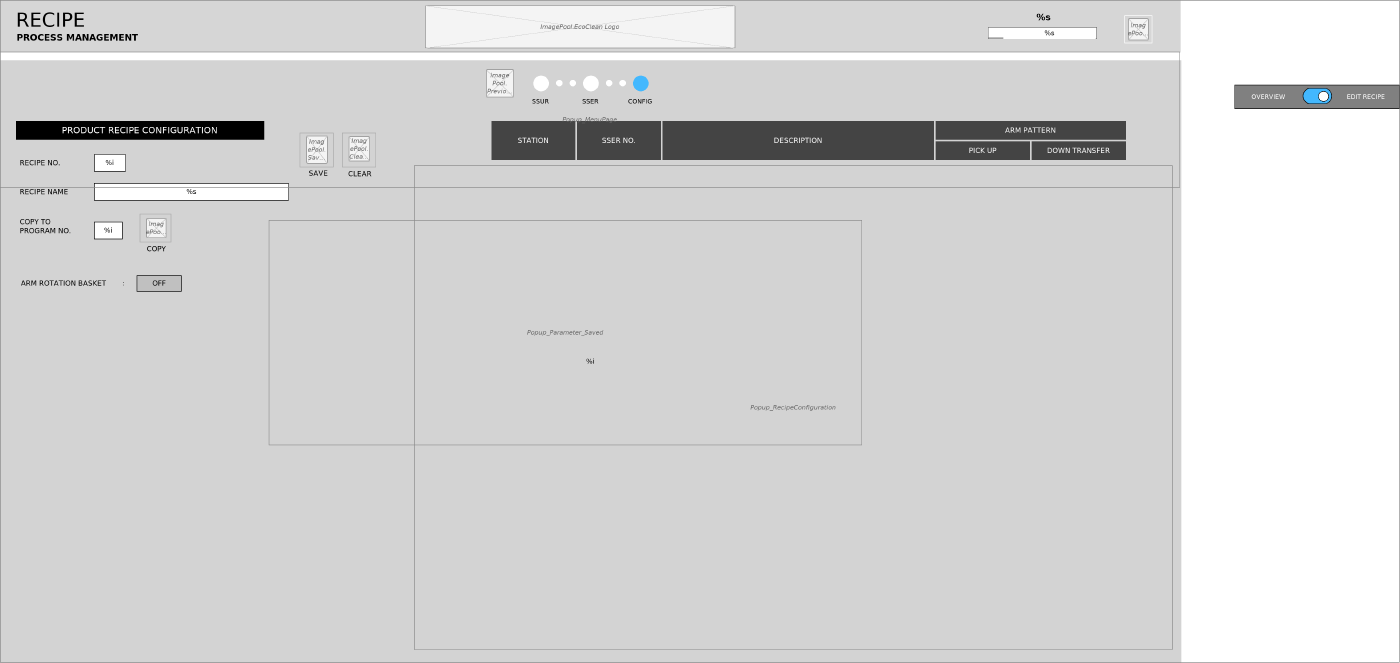
VISUALIZATION RecipeConfiguration_Page  // 2276x1079
    RoundedRectangle (245,275 1437x791)
    Rectangle (0,98 1920x981), "%i", text variable: Global_Variables_Arm_Persistent.DSA1fbPnpSequenceMemoryStore.iProductRecipeNo
    Rectangle (0,63 1920x26)
        p3528305787: HMI_Ctrl.ANIMATION3
    Rectangle (0,0 1919x85)
    Group (23,6 321x67)
        Label (0,0 267x53), "RECIPE"
        Label (1,43 320x24), "PROCESS MANAGEMENT"
    Frame (673,269 1233x788)
        shows Popup_RecipeConfiguration()
    Rectangle (799,197 136x63), "STATION"
    Rectangle (938,197 136x63), "SSER NO."
    Rectangle (1077,197 441x63), "DESCRIPTION"
    Group (1521,197 309x63)
        Rectangle (0,33 153x30), "PICK UP"
        Rectangle (156,33 153x30), "DOWN TRANSFER"
        Rectangle (0,0 309x30), "ARM PATTERN"
    Group (1828,25 45x45)
        OnMouseClick: toggle HMI_Ctrl.MenuButton
        RoundedRectangle (0,0 45x45), colour toggle: HMI_Ctrl.MenuButton
        Image (6,5 33x35), image: ImagePool.Menu Button
    Group (2007,137 269x41)
        RoundedRectangle (0,1 269x39)
        Label (1,0 108x41), "OVERVIEW"
        Label (161,0 105x41), "EDIT RECIPE"
        Group (111,6 47x26)
            OnMouseClick: change screen: Recipe_Page
            Group (0,0 47x26)
                Ellipse (0,0 26x26)
                Ellipse (21,0 26x26)
                RoundedRectangle (8,0 29x26)
            Ellipse (1,1 24x24)
            Ellipse (23,1 23x24)
            RoundedRectangle (9,1 28x24)
            Ellipse (25,5 17x17)
    Ellipse (867,123 25x25)
    Ellipse (948,123 25x25)
    Ellipse (904,130 10x10)
    Ellipse (926,130 10x10)
    Ellipse (985,130 10x10)
    Ellipse (1007,130 10x10)
    Ellipse (1029,123 25x25)
    Label (847,153 64x24), "SSUR"
    Label (928,153 64x24), "SSER"
    Label (1009,153 64x24), "CONFIG"
    Image (790,113 45x45), image: ImagePool.Previous Button
        OnMouseClick: change screen: RecipeSSER_Page
    Rectangle (26,197 403x30), "PRODUCT RECIPE CONFIGURATION"
    Label (29,253 93x24), "RECIPE NO."
    RoundedRectangle (153,251 51x28), "%i", text variable: Global_Variables_Arm_Persistent.DSA1fbPnpSequenceMemoryStore.iProductRecipeNo
        OnMouseDown: write the text variable via Default, min 1, max 40
    Label (29,300 101x24), "RECIPE NAME"
    RoundedRectangle (153,298 316x28), "%s", text variable: Global_Variables_Arm_Persistent.DSA1fbPnpSequenceMemoryStore.DsA1inPnpSequenceMemory.sDescription
        OnMouseDown: write the text variable via VisuDialogs.Keypad
    Label (29,348 110x41), "COPY TO PROGRAM NO."
    RoundedRectangle (153,361 46x28), "%i", text variable: DSA1fbPnpSequenceMemoryStore.iCopyToProductRecipeNo
        OnMouseDown: write the text variable via VisuDialogs.Numpad, min 1, max 40
    Image (691,9 504x69), image: ImagePool.EcoClean Logo
    Group (227,348 51x69), invisible if: bMainOnOff
        Label (6,45 42x24), "COPY"
        RoundedRectangle (0,0 51x46), colour toggle: DSA1fbPnpSequenceMemoryStore.bCopyPB
            tap DSA1fbPnpSequenceMemoryStore.bCopyPB
        Image (11,7 32x32), image: ImagePool.Copy Button
            OnMouseDown: execute { DSA1fbPnpSequenceMemoryStore.bCopyPB:=1; }
            OnMouseUp: execute { DSA1fbPnpSequenceMemoryStore.bCopyPB:=0; }
    Group (1606,17 179x46)
        Button (0,27 177x19), image: VisuSymbols.Symbols.AddUser
        Rectangle (25,28 150x18), "%s", text variable: fbHmiTF1800_UserlevelManagement.dsHmiUserStatus_Active.sLoginName
        Rectangle (2,0 177x22), "%s", text variable: DSLocalSystemTimeML.sCurrentDT24Hr_General
    Group (487,216 56x80), invisible if: bMainOnOff
        Label (5,52 51x28), "SAVE", invisible if: bMainOnOff
        RoundedRectangle (0,0 55x56), colour toggle: bRecipeSavePb
            tap bRecipeSavePb
        Image (11,5 34x45), image: ImagePool.Save Button
            OnMouseDown: execute { bRecipeSavePb:=1; }
            OnMouseUp: execute { bRecipeSavePb:=0; }
    Frame (437,358 964x366), invisible if: NOT stWritePersistentData.SaveHR
        shows Popup_Parameter_Saved()
    Label (31,449 183x24), "ARM ROTATION BASKET"
    Label (196,449 19x24), ":"
    Rectangle (222,448 73x26), "ON", invisible if: NOT DSA1fbPnpSequenceMemoryStore.DsA1inPnpSequenceMemory.bArmRotaryBarrelEnable
        OnMouseDown: execute { DSA1fbPnpSequenceMemoryStore.DsA1inPnpSequenceMemory.bArmRotaryBarrelEnable:=FALSE; }
    Rectangle (222,448 73x26), "OFF", invisible if: DSA1fbPnpSequenceMemoryStore.DsA1inPnpSequenceMemory.bArmRotaryBarrelEnable
        OnMouseDown: execute { DSA1fbPnpSequenceMemoryStore.DsA1inPnpSequenceMemory.bArmRotaryBarrelEnable:=TRUE; }
    Label (560,271 50x24), "CLEAR"
    RoundedRectangle (556,216 55x56), colour toggle: bProductRecipeClearPb
        tap bProductRecipeClearPb
    Image (567,222 34x40), image: ImagePool.Clear Button
        OnMouseDown: execute { bProductRecipeClearPb:=1; }
        OnMouseUp: execute { bProductRecipeClearPb:=0; }
    Frame (0,84 1918x221), invisible if: HMI_Ctrl.CloseMenuButton
        shows Popup_MenuPage()
END_VISUALIZATION

(* stored: Version 1.1.0.1, ProductVersion 3.1.4024.12
   Visu RecipeConfiguration_Page: Id {65deb92a-ed8e-49f0-a059-b617d6bd91ff} *)
